// TIA Portal V17 export
// export: Created 2025-06-26T06:49:28.4878614Z, ExportSetting WithDefaults, DisplayName Totally Integrated Automation Portal, DisplayVersion V17 Update 8, DisplayName TIA Portal Openness, DisplayVersion V17 Update 8, DisplayName TIA Portal Version Control Interface, DisplayVersion V17, DisplayName STEP 7 Professional, DisplayVersion V17 Update 8, DisplayName STEP 7 Safety, DisplayVersion V17 Update 6, DisplayName WinCC Advanced, DisplayVersion V17 Update 8
TYPE "stABB_ACSx80_Tx"
// stored: IsFailsafeCompliant false
   STRUCT
      CW : Word;   // Command word (58.101)
      Ref1 : Word;   // Reference 1 (58.102)
      Ref2 : Word;   // Reference 2 (58.103)
      DataIO_4 : Word;   // User configurable 1 (58.104)
      DataIO_5 : Word;   // User configurable 2 (58.105)
      DataIO_6 : Word;   // User configurable 3 (58.106)
      DataIO_7 : Word;   // User configurable 4 (58.107)
      DataIO_8 : Word;   // User configurable 5 (58.108)
   END_STRUCT;
END_TYPE
